KUKA KRL program: chk_w8_wechs_ok.src

&ACCESS RVO12
&REL 8
&COMMENT Check tool change
DEF chk_w8_wechs_ok( )
;177 => wkz1 C1
;185 => wkz2 C2
;161 => wkz3 GRIPER ACTROS
;169 => wkz4 GRIPER ACELO
;193 => wkz5 C3
;201 => wkz6 GRIPER AXOR/ATEGO
;219 => ACOPLAMENTO OK
;3320=> GRIPER NA ST600
; VERIFICAÇÃO DE FERRAMENTA: TOOL CHANGE

WAIT FOR ((($in[161]) OR (NOT ($in[161]) and ($in[3320]))) AND (($in[169]) OR (NOT ($in[169]) and ($in[3320]))) AND ($in[177]) AND ($in[185]) AND ($in[193]) AND (($in[201]) or (not ($in[201]) and ($in[3320]))) AND (NOT $in[219]))


END
